// TIA Portal V18 export
DATA_BLOCK "НулевыеБлокировки_DB"   // DB56
VERSION : 0.1
// stored: AutoNumber true, DBAccessibleFromOPCUA true, InstanceOfName НулевыеБлокировки, InstanceOfType FB
"НулевыеБлокировки"
   // VAR_INPUT
   //    x_Nok : Bool;
   // END_VAR
   // VAR_OUTPUT
   //    y_ERROR : Bool;
   // END_VAR
   // VAR_IN_OUT
   //    ton_delay : Time;
   // END_VAR
   // VAR
   //    IEC_Timer_0_Instance { S7_SetPoint := 'True'} : TON_TIME;
   // END_VAR
BEGIN
END_DATA_BLOCK
